PROGRAM analogSignals_ex05
VAR
	rpmcontrol			: REAL;
	rpm					: REAL;
	
	LIN_TRAFO 			: FB_Scale;
END_VAR

LIN_TRAFO(
	fIN:= rpmcontrol, 
	fIN_min:= 0, 
	fIN_max:= 120, 
	fOUT_min:= 4, 
	fOUT_max:= 20, 
	fOUT=> rpm);

END_PROGRAM

(* stored: Version 1.1.0.1
   POU analogSignals_ex05: Id {7dec8ca8-615b-45b9-835c-4212b8af76d4}, SpecialFunc None *)
